Fanuc KAREL source: ko00106.KL

-- PROVISIONAL review KL for V940-1; original PC SHA256 9707abb740dbe8d9ec98bd9ea6dc4d66034fde168acfe167cf658260282dd6dd
-- Incomplete behavior may be omitted. Consult companion uncertainty JSON. Do not deploy.
PROGRAM KO00106
%NOLOCKGROUP
VAR
  A : REAL
  B : INTEGER
  OUT : REAL
BEGIN
  -- V9_ZERO_TABLE_METADATA_HINT layout=0001; no indexed target words; source/name/runtime held
  -- UNRESOLVED_PC offsets 5-13; opcodes 9D,64,23
  -- UNRESOLVED_PC offsets 18-29; opcodes 2E,23
  -- UNRESOLVED_PC offsets 34-57; opcodes 27,22,27,21,64,76,23
  -- UNRESOLVED_PC offsets 62-66; opcodes 7F
END KO00106
